// TIA Portal V18 export
DATA_BLOCK "Faults&warnings"   // DB67
{ S7_Optimized_Access := 'TRUE' }
VERSION : 0.1
// stored: AutoNumber true, DBAccessibleFromOPCUA true, IsOnlyStoredInLoadMemory false, IsRetainMemResEnabled false, IsWriteProtectedInAS false, MemoryReserve 100
   VAR
      "Critical Alarm Metering A" : Bool;
      "Critical Alarm metering B" : Bool;
      "Critical Alarm metering A&B" : Bool;
      "alarm Level" : Int;
      "Alarm popped" : Bool;
      "Alarm Number" : Int;
      "Alarm ack Hmi" : Bool;
      "Alarm class" : Int;
      "Fault display register" : Int;
      "Fault display register Moved" : Int;
      "Fault present" : Bool;
      "Status Nok" : Struct
         "Drive controller A NK" : Bool;
         "Drive controller B NK" : Bool;
         "Agitator A Fault" : Bool;
         "Agitator B Fault" : Bool;
         "Mixer Drive NK" : Bool;
         "Pressure sensor Pump A Inlet" : Bool;
         "Pressure Sensor Pump B Inlet" : Bool;
         "Pressure sensor Pump A Outlet" : Bool;
         "Pressure Sensor Pump B Outlet" : Bool;
         "Over pressure A inlet" : Bool;
         "Over pressure B inlet" : Bool;
         "Over pressure A outlet" : Bool;
         "Over pressure B outlet" : Bool;
         "Emergency stop" : Bool;
         "Control ON" : Bool;
         "Pressure sensor vessel A1" : Bool;
         "Pressure sensor vessel A2" : Bool;
         "Pressure sensor vessel B1" : Bool;
         "Pressure sensor vessel B2" : Bool;
         "Material Supply A" : Bool;
         "Material Supply B" : Bool;
         "Low level B2" : Bool;
         "Level Empty B2" : Bool;
         "Level sensor B2" : Bool;
         "Low level A1" : Bool;
         "Level empty A1" : Bool;
         "Level Sensor Pressure vessel A" : Bool;
         "Low level A2" : Bool;
         "Level empty A2" : Bool;
         "Low level B1" : Bool;
         "Level empty B1" : Bool;
         "Level Sensor Pressure vessel B" : Bool;
         "Flowrate error" : Bool;
         "Level Low Pressure Vessel A" : Bool;
         "Level Low Pressure Vessel B" : Bool;
         "Level Empty Pressure Vessel A" : Bool;
         "Level Empty Pressure Vessel B" : Bool;
         "Level Low Catridge A" : Bool;
         "Level Low Catridge B" : Bool;
         "Level Empty Catridge A" : Bool;
         "Level Empty Catridge B" : Bool;
         "Level Low Drum A1" : Bool;
         "Level Low Drum B1" : Bool;
         "Level Low Drum A2" : Bool;
         "Level Low Drum B2" : Bool;
         "Level Empty Drum A1" : Bool;
         "Level Empty Drum B1" : Bool;
         "Level Empty Drum A2" : Bool;
         "Level Empty Drum B2" : Bool;
      END_STRUCT;
      "Operator message 1" : Int;
      "Operator message 2" : Int;
      "alarm popped out" : Bool;
      "faultnumber in hmi" : Int;
      "alarm Display number" : Int;
      "Current Scroll Number" : DInt := 1;
   END_VAR
BEGIN
END_DATA_BLOCK
